(* IEC 61131-3 sources: Lasal/CPU_5344_V01/Class/sawToolSettingsMpsControl, 1 file *)

(* ---- sawToolSettingsMpsControl.st ---- *)
(*!
<Class
	Name               = "sawToolSettingsMpsControl"
	Revision           = "1.0"
	RealtimeTask       = "false"
	CyclicTask         = "false"
	BackgroundTask     = "false"
	Sigmatek           = "false"
	OSInterface        = "false"
	HighPriority       = "false"
	Automatic          = "false"
	UpdateMode         = "Prescan"
	SharedCommandTable = "true"
	Objectsize         = "(284,120)">
	<Channels>
		<Server Name="setting1" Visualized="true" Initialize="false" WriteProtected="false" Retentive="false" Comment="min. sawing angle (in 1/10 degree) where 90 degree is right angled "/>
		<Server Name="setting2" Visualized="true" Initialize="false" WriteProtected="false" Retentive="false" Comment="max. sawing angle (in 1/10 degree) where 90 degree is right angled"/>
		<Client Name="iMaxAngle" Required="true" Internal="false"/>
		<Client Name="iMinAngle" Required="true" Internal="false"/>
	</Channels>
	<Network Name="sawToolSettingsMpsControl">
		<!-- List of Components in this network -->
		<Components>
			<Object
				Name       = "_base"
				Class      = "baseToolSettingsMpsControl"
				Position   = "(218,120)"
				Visualized = "true">
				<Channels>
					<Server Name="amountOfSettings" Value="4"/>
					<Server Name="ClassSvr"/>
					<Server Name="Name"/>
					<Server Name="plane"/>
					<Server Name="toolType" Value="1"/>
				</Channels>
			</Object>
		</Components>
		<Comments>
		</Comments>
		<!-- List of Connections in this network -->
		<Connections>
			<Connection Source="this.ClassSvr" Destination="_base.ClassSvr" Vertices="(690,210),(518,210),"/>
			<Connection Source="this.toolType" Destination="_base.toolType" Vertices="(690,270),(518,270),"/>
			<Connection Source="this.amountOfSettings" Destination="_base.amountOfSettings" Vertices="(690,450),(518,450),"/>
			<Connection Source="this.plane" Destination="_base.plane" Vertices="(690,390),(518,390),"/>
			<Connection Source="this.Name" Destination="_base.Name" Vertices="(690,330),(518,330),"/>
		</Connections>
		<!-- Headerfiles -->
		<Options>
		</Options>
	</Network>
</Class>
*)
#pragma using baseToolSettingsMpsControl

sawToolSettingsMpsControl : CLASS
: baseToolSettingsMpsControl
  //Servers:
	setting1 	: SvrCh_DINT;
	setting2 	: SvrCh_DINT;
  //Clients:
	iMinAngle 	: CltCh_DINT;
	iMaxAngle 	: CltCh_DINT;
  //Variables:
  //Functions:

	FUNCTION VIRTUAL GLOBAL setting1::Read
		VAR_OUTPUT
			output (EAX) 	: DINT;
		END_VAR;

	FUNCTION VIRTUAL GLOBAL setting2::Read
		VAR_OUTPUT
			output (EAX) 	: DINT;
		END_VAR;
  //Tables:
	FUNCTION @STD
		VAR_OUTPUT
			ret_code	: CONFSTATES;
		END_VAR;
	FUNCTION GLOBAL TAB @CT_;
END_CLASS;

// JdK 4-2-2020: sawToolSettingsMpsControl created for first test to read in settings to pc
// at this moment the class is only for storage off fixed machine data for saw tools

FUNCTION VIRTUAL GLOBAL sawToolSettingsMpsControl::setting1::Read
	VAR_OUTPUT
		output (EAX) 	: DINT;
	END_VAR

  iMinAngle:=iMinAngle.Read();
  setting1:= iMinAngle;

	output := setting1;

END_FUNCTION

FUNCTION VIRTUAL GLOBAL sawToolSettingsMpsControl::setting2::Read
	VAR_OUTPUT
		output (EAX) 	: DINT;
	END_VAR

  iMaxAngle:=iMaxAngle.Read();
  setting2:= iMaxAngle;

	output := setting2;

END_FUNCTION
